PROGRAM INTERNAL Clock
// RTC - Real time clock low precision synchronizable with NTS
// TickClocl - Hi presition from start of the system

END_PROGRAM

(* stored: Version 1.1.0.1, ProductVersion 3.1.4024.6
   POU Clock: Id {cd04d6fc-8735-001f-16e8-7e49bd4514a9}, SpecialFunc None *)
